FUNCTION_BLOCK T_ExternalControllerMock IMPLEMENTS I_PackML_ExternalController
VAR_INPUT
END_VAR
VAR_OUTPUT
	_newState	: Tc3_PackML_V2.E_PMLCommand;
END_VAR
VAR

END_VAR

{warning 'add property implementation'}
PROPERTY Control : I_PackML_Control
SET
END_SET
END_PROPERTY

METHOD ModeChanged
VAR_INPUT
	NewMode	: E_PMLUnitMode;
END_VAR
END_METHOD

METHOD StateChanged
VAR_INPUT
	NewState	: Tc3_PackML_V2.E_PMLCommand;
END_VAR
_newState := NewState;
END_METHOD

END_FUNCTION_BLOCK

(* stored: Version 1.1.0.1, ProductVersion 3.1.4024.12
   POU T_ExternalControllerMock: Id {43aa55ca-47db-4640-96c7-f6db5856e5d2}, SpecialFunc None
   Property Control: Id {c1ab2343-083b-4a20-9bc7-63b337d93079}
   Set Set: Id {2105b7ce-a4fe-45eb-b906-805c1820e865}
   Method ModeChanged: Id {edcda9d9-d9d0-46c2-8523-9d1e40c4b24d}
   Method StateChanged: Id {99b3c0a7-a033-4b9e-84ef-400e8952a4d2} *)
